FUNCTION_BLOCK T_Assertion
VAR_INPUT
END_VAR
VAR_OUTPUT
END_VAR
VAR
    _AssertionFailed : BOOL;
    _AssertionMessage : T_MaxString;
    _ExpectedAsString : T_MaxString;
    _ActualAsString   : T_MaxString;
END_VAR

METHOD AssertEquals_BOOL : BOOL;
VAR_INPUT
    Source   : T_MaxString;
    Expected : BOOL;
    Actual   : BOOL;
    Message  : T_MaxString;
END_VAR
IF Expected <> Actual THEN
    F_LogResult(Source, F_FormatStringEx1('Assertion Failed - %s', Message));
    RETURN;
END_IF

AssertEquals_BOOL := TRUE;
END_METHOD

METHOD AssertEquals_DINT : BOOL
VAR_INPUT
    Source   : T_MaxString;
    Expected : DINT;
    Actual   : DINT;
    Message  : T_MaxString;
END_VAR
IF Expected <> Actual THEN
    F_LogResult(Source, F_FormatStringEx1('Assertion Failed - %s', Message));
END_IF

AssertEquals_DINT := TRUE;
END_METHOD

METHOD AssertEquals_STRING : BOOL
VAR_INPUT
    Source   : T_MaxString;
    Expected : T_MaxString;
    Actual   : T_MaxString;
    Message  : T_MaxString;
END_VAR
IF Expected <> Actual THEN
    F_LogResult(Source, F_FormatStringEx1('Assertion Failed - %s', Message));
END_IF

AssertEquals_STRING := TRUE;
END_METHOD

PROPERTY AssertionFailed : BOOL
GET
AssertionFailed := _AssertionFailed;
END_GET
END_PROPERTY

PROPERTY AssertionMessage : T_MaxString
GET
AssertionMessage := _AssertionMessage;
END_GET
END_PROPERTY

END_FUNCTION_BLOCK

(* stored: Version 1.1.0.1, ProductVersion 3.1.4024.12
   POU T_Assertion: Id {a1aef330-5110-4c04-a4ca-af23774823fc}, SpecialFunc None
   Folder Methods: Id {b5309a9f-d22b-4798-ac38-129f27945b0a}
   Folder Properties: Id {2b96df32-c9bc-482b-8e63-e4930a06246e}
   Method AssertEquals_BOOL: Id {cdb21bbb-0bd7-498a-af51-940faf207ee6}
   Method AssertEquals_DINT: Id {87caa963-e045-4af5-b563-b93e89f13ab7}
   Method AssertEquals_STRING: Id {bc26e0ad-c421-4d8e-b875-daeab2504431}
   Property AssertionFailed: Id {efe5b392-bd52-4186-adc6-a08baeb9456e}
   Get Get: Id {58033276-2b54-4cf0-846a-6cb8d1dec6d1}
   Property AssertionMessage: Id {450e3501-7d12-45c4-a5bf-d12c3afea520}
   Get Get: Id {fe321a98-402a-43fe-9184-70844f27500e} *)
